// TIA Portal V17 export
// export: Created 2022-07-20T06:59:45.2265641Z, ExportSetting WithDefaults, DisplayName Totally Integrated Automation Portal, DisplayVersion V17, DisplayName TIA Portal Openness, DisplayVersion V17, DisplayName TIA Portal Version Control Interface, DisplayVersion V17, DisplayName SINAMICS Startdrive Advanced, DisplayVersion V17, DisplayName SINAMICS Startdrive G130, G150, S120, S150, SINAMICS MV, S210, DisplayVersion V17, DisplayName SINAMICS Startdrive G110M, G120, G120C, G120D, G120P, G115D, DisplayVersion V17, DisplayName STEP 7 Professional, DisplayVersion V17, DisplayName STEP 7 Safety, DisplayVersion V17, DisplayName WinCC Advanced, DisplayVersion V17
FUNCTION_BLOCK "FB10091_HeatingResistanceControl"   // FB10091, LAD
TITLE = FB10091_HeatingResistanceControl
{ S7_Optimized_Access := 'TRUE' }
AUTHOR : Jonathan
FAMILY : 1009x_DRYER_UV
VERSION : 1.0
// Release note
// 1.0 - Feature developped
// stored: AutoNumber false, IsIECCheckEnabled false, IsRetainMemResEnabled false, MemoryReserve 100, SetENOAutomatically false, UDAEnableTagReadback false
   VAR_INPUT
      EnableModule : Bool;
      PowerOK : Bool;
      StartHeatingCommand : Bool;
   END_VAR
   VAR_OUTPUT
      StartHeatingSignal : Bool;
      ActivePowerRelay : Bool;
   END_VAR
   VAR
      TOF_MaintainAfterStop { S7_SetPoint := 'True'} : TOF_TIME;
   END_VAR
BEGIN

REGION Network 1: Active power relay
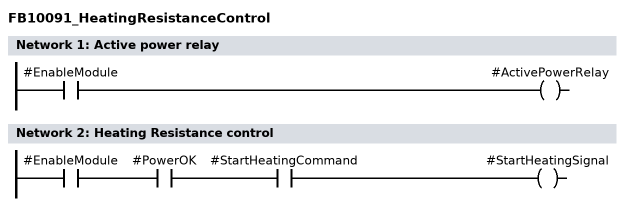
   RUNG wire#powerrail
      Contact( #EnableModule )
      Coil( #ActivePowerRelay )
   END_RUNG
   // the same network as SCL:
   #ActivePowerRelay := #EnableModule;
END_REGION

REGION Network 2: Heating Resistance control
   RUNG wire#powerrail
      Contact( #EnableModule )
      Contact( #PowerOK )
      Contact( #StartHeatingCommand )
      Coil( #StartHeatingSignal )
   END_RUNG
   // the same network as SCL:
   #StartHeatingSignal := #EnableModule AND #PowerOK AND #StartHeatingCommand;
END_REGION
END_FUNCTION_BLOCK
